FUNCTION BITS_TO_WORD
  (* Standard: 61499-1 *)
  (* Version 1.0, 2024-02-22, franz *)
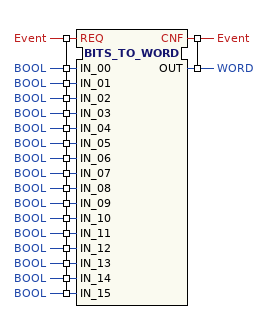
  EVENT_INPUT
    REQ WITH IN_00, IN_01, IN_02, IN_03, IN_04, IN_05, IN_06, IN_07, IN_08, IN_09, IN_10, IN_11, IN_12, IN_13, IN_14, IN_15;
  END_EVENT
  EVENT_OUTPUT
    CNF WITH OUT;
  END_EVENT
  VAR_INPUT
    IN_00 : BOOL; (* BIT 00 *)
    IN_01 : BOOL; (* BIT 01 *)
    IN_02 : BOOL; (* BIT 02 *)
    IN_03 : BOOL; (* BIT 03 *)
    IN_04 : BOOL; (* BIT 04 *)
    IN_05 : BOOL; (* BIT 05 *)
    IN_06 : BOOL; (* BIT 06 *)
    IN_07 : BOOL; (* BIT 07 *)
    IN_08 : BOOL; (* BIT 08 *)
    IN_09 : BOOL; (* BIT 09 *)
    IN_10 : BOOL; (* BIT 10 *)
    IN_11 : BOOL; (* BIT 11 *)
    IN_12 : BOOL; (* BIT 12 *)
    IN_13 : BOOL; (* BIT 13 *)
    IN_14 : BOOL; (* BIT 14 *)
    IN_15 : BOOL; (* BIT 15 *)
  END_VAR
  VAR_OUTPUT
    OUT : WORD; (* WORD Output *)
  END_VAR
  BODY IN ST:
FUNCTION BITS_TO_WORD

VAR_INPUT
	IN_00 : BOOL;    // BIT 00
	IN_01 : BOOL;    // BIT 01
	IN_02 : BOOL;    // BIT 02
	IN_03 : BOOL;    // BIT 03
	IN_04 : BOOL;    // BIT 04
	IN_05 : BOOL;    // BIT 05
	IN_06 : BOOL;    // BIT 06
	IN_07 : BOOL;    // BIT 07
	IN_08 : BOOL;    // BIT 08
	IN_09 : BOOL;    // BIT 09
	IN_10 : BOOL;    // BIT 10
	IN_11 : BOOL;    // BIT 11
	IN_12 : BOOL;    // BIT 12
	IN_13 : BOOL;    // BIT 13
	IN_14 : BOOL;    // BIT 14
	IN_15 : BOOL;    // BIT 15
END_VAR

VAR_OUTPUT
	OUT : WORD;    // WORD Output
END_VAR

(* this Function combines the 16 Bits to a word *)
OUT.0 := IN_00;
OUT.1 := IN_01;
OUT.2 := IN_02;
OUT.3 := IN_03;
OUT.4 := IN_04;
OUT.5 := IN_05;
OUT.6 := IN_06;
OUT.7 := IN_07;
OUT.8 := IN_08;
OUT.9 := IN_09;
OUT.10 := IN_10;
OUT.11 := IN_11;
OUT.12 := IN_12;
OUT.13 := IN_13;
OUT.14 := IN_14;
OUT.15 := IN_15;

END_FUNCTION
  END_BODY
END_FUNCTION
